TYPE ST_SDI_6_0 :
(**************************************************************************************
 * 	Application		:	BoxControl Framework
 *	Revision		:	$Revision: 404529 $
 *	Revision date	:	$Date: 2018-04-23 08:21:38 +0200 (Mo., 23 Apr 2018) $
 *	Last changed by	:	$Author: b7bolm $
 *	URL				:	$URL: http://almscdc.swisslog.com/repo/SWPD/Development/BoxControlFramework/20_Release/trunk/01_Software/BCF/BCF/JumpStart/20_Product/10_App/11_Com/10_Lib/10_Conv/12_MFCS/11_SIS/01_DUTs/10_SIS_6_0/ST_SDI_6_0.TcDUT $
 *
 *	Purpose			:	SDI Structure
 *
 * ------------------------------------------------------------------------------------
 *	Copyright Swisslog [IP AG], Switzerland. All rights reserved.
 * 
 * ------------------------------------------------------------------------------------
 *	
 * 	Revision History: 
 *
 * 	VERSION			DATE			INITIALS			DESCRIPTION
 *	0.1				01.01.2001		swl					Example
 *
 **************************************************************************************)
STRUCT
	SignalNumber	: STRING(SIS_6_0.SDI_SIGNALNUMBER_STRINGLENGTH); // 4 Digit Signal Number 
	SignalState		: STRING(SIS_6_0.SDI_SIGNALSTATE_STRINGLENGTH); // 1 Digit Signal Status 
	ReturnCode		: STRING(SIS_6_0.ERRORCODE_STRINGLENGTH) := '0000'; // 4 Digit Return Code 
END_STRUCT
END_TYPE

(* stored: Version 1.1.0.1, ProductVersion 3.1.4022.12
   DUT ST_SDI_6_0: Id {75db16b6-b649-4186-8579-a8e8b6617fe9} *)
